Staubli VAL3: goHome.pgx

program goHome()
begin
  // go to HOME
  // check if the robot is not in cycle
  if !(cycleStatus:bCycle or cycleStatus:bSimulation)
    cycleStatus:bToHome=true
    watch(cycleStatus:bToHome==false,3)
    // wait end of HOME
    watch(cycleStatus:bIsHome,3)
    waitEndMove()
    watch(cycleStatus:bSimulation==false,3)
  endIf
end
